// TIA Portal V20 export
TYPE "LBP_typeAlarmMsgs"
TITLE = PLC-Error / Messages / Erreur AP / messages
// User data type for block LBP_AlarmMessage [DB2] / Type de données utilisateur pour bloc LBP_AlarmMessage [DB2]
   STRUCT
      Chan : Array[1..10] of Struct   // From Channel 1..10 / Depuis canal 1..10
         FDD : Array[0..15] of Bool;   // Feed disable / Désactiver avance
         RID : Array[0..15] of Bool;   // Read-in disable / Désactiver importation
         NCSD : Array[0..15] of Bool;   // NC start disable / Désactiver Départ CN
         FdStop_1 : Array[0..15] of Bool;   // Feed stop GEOaxis 1 / Arrêt avance axe GEO 1
         FdStop_2 : Array[0..15] of Bool;   // Feed stop GEOaxis 2 / Arrêt avance axe GEO 2
         FdStop_3 : Array[0..15] of Bool;   // Feed stop GEOaxis 3 / Arrêt avance axe GEO 3
      END_STRUCT;
      Axis : Array[1..31] of Struct   // From Axis 1..31 / Depuis axe 1..31
         FdStop : Array[0..15] of Bool;   // Feed stop axis/spindle / Arrêt avance axe/broche
      END_STRUCT;
      AddValUserA0 : Array[0..63] of Int;   // Additional value for alarms in the user area 0 (700000..700063) / Valeur additionnelle pour les alarmes dans la zone utilisateur 0 (700000..700063)
      ChanA : Array[1..10] of Struct   // From Channel 1..10 / Depuis canal 1..10
         FDD_5C00xx : Array[0..15] of Bool;   // Feed disable Alarm no. 5C0000..5C0015 / Désactiver avance Alarme n° 5C0000..5C0015
         FDD_RID_5C01xx : Array[0..31] of Bool;   // Feed and read-in disable Alarm no. 5C0100..5C0131 / Désactiver avance et importation Alarme n° 5C0100..5C0131
         RID_5C02xx : Array[0..31] of Bool;   // Read-in disable Alarm no. 5C0200..5C0231 / Désactiver avance Alarme n° 5C0200..5C0231
         NCSD_5C03xx : Array[0..15] of Bool;   // NC start disable Alarm no. 5C0300..5C0315 / Désactiver Départ CN Alarme n° 5C0300..5C0315
         FdStop_1_5C11xx : Array[0..15] of Bool;   // Feed stop GEOaxis 1 Alarm no. 5C1100..5C1115 / Arrêt avance axe GEO 1 Alarme n° 5C1100..5C1115
         FdStop_2_5C12xx : Array[0..15] of Bool;   // Feed stop GEOaxis 2 Alarm no. 5C1200..5C1215 / Arrêt avance axe GEO 2 Alarme n° 5C1200..5C1215
         FdStop_3_5C13xx : Array[0..15] of Bool;   // Feed stop GEOaxis 3 Alarm no. 5C1300..5C1315 / Arrêt avance axe GEO 3 Alarme n° 5C1300..5C1315
      END_STRUCT;
      AxisA : Array[1..31] of Struct   // From Axis 1..31 / Depuis axe 1..31
         AAFdStop60AAxx : Array[0..15] of Bool;   // Feed stop axis/spindle / Arrêt avance axe/broche
      END_STRUCT;
      res552 : Word;   // Reserved / Réservé
      UserA : Array[0..63] of Struct
         A70UUxx : Array[0..63] of Bool;   // Alarm 70UU00..70UU63 (user area) / Alarme 70UU00..70UU63 (zone utilisateur)
      END_STRUCT;
   END_STRUCT;
   // // Chan[2].FDD : Feed disable / Désactiver avance
   // // Chan[3].FDD : Feed disable / Désactiver avance
   // // Chan[4].FDD : Feed disable / Désactiver avance
   // // Chan[5].FDD : Feed disable / Désactiver avance
   // // Chan[6].FDD : Feed disable / Désactiver avance
   // // Chan[7].FDD : Feed disable / Désactiver avance
   // // Chan[8].FDD : Feed disable / Désactiver avance
   // // Chan[9].FDD : Feed disable / Désactiver avance
   // // Chan[10].FDD : Feed disable / Désactiver avance
   // // Chan[2].RID : Read-in disable / Désactiver importation
   // // Chan[3].RID : Read-in disable / Désactiver importation
   // // Chan[4].RID : Read-in disable / Désactiver importation
   // // Chan[5].RID : Read-in disable / Désactiver importation
   // // Chan[6].RID : Read-in disable / Désactiver importation
   // // Chan[7].RID : Read-in disable / Désactiver importation
   // // Chan[8].RID : Read-in disable / Désactiver importation
   // // Chan[9].RID : Read-in disable / Désactiver importation
   // // Chan[10].RID : Read-in disable / Désactiver importation
   // // Chan[2].NCSD : NC start disable / Désactiver Départ CN
   // // Chan[3].NCSD : NC start disable / Désactiver Départ CN
   // // Chan[4].NCSD : NC start disable / Désactiver Départ CN
   // // Chan[5].NCSD : NC start disable / Désactiver Départ CN
   // // Chan[6].NCSD : NC start disable / Désactiver Départ CN
   // // Chan[7].NCSD : NC start disable / Désactiver Départ CN
   // // Chan[8].NCSD : NC start disable / Désactiver Départ CN
   // // Chan[9].NCSD : NC start disable / Désactiver Départ CN
   // // Chan[10].NCSD : NC start disable / Désactiver Départ CN
   // // Chan[2].FdStop_1 : Feed stop GEOaxis 1 / Arrêt avance axe GEO 1
   // // Chan[3].FdStop_1 : Feed stop GEOaxis 1 / Arrêt avance axe GEO 1
   // // Chan[4].FdStop_1 : Feed stop GEOaxis 1 / Arrêt avance axe GEO 1
   // // Chan[5].FdStop_1 : Feed stop GEOaxis 1 / Arrêt avance axe GEO 1
   // // Chan[6].FdStop_1 : Feed stop GEOaxis 1 / Arrêt avance axe GEO 1
   // // Chan[7].FdStop_1 : Feed stop GEOaxis 1 / Arrêt avance axe GEO 1
   // // Chan[8].FdStop_1 : Feed stop GEOaxis 1 / Arrêt avance axe GEO 1
   // // Chan[9].FdStop_1 : Feed stop GEOaxis 1 / Arrêt avance axe GEO 1
   // // Chan[10].FdStop_1 : Feed stop GEOaxis 1 / Arrêt avance axe GEO 1
   // // Chan[2].FdStop_2 : Feed stop GEOaxis 2 / Arrêt avance axe GEO 2
   // // Chan[3].FdStop_2 : Feed stop GEOaxis 2 / Arrêt avance axe GEO 2
   // // Chan[4].FdStop_2 : Feed stop GEOaxis 2 / Arrêt avance axe GEO 2
   // // Chan[5].FdStop_2 : Feed stop GEOaxis 2 / Arrêt avance axe GEO 2
   // // Chan[6].FdStop_2 : Feed stop GEOaxis 2 / Arrêt avance axe GEO 2
   // // Chan[7].FdStop_2 : Feed stop GEOaxis 2 / Arrêt avance axe GEO 2
   // // Chan[8].FdStop_2 : Feed stop GEOaxis 2 / Arrêt avance axe GEO 2
   // // Chan[9].FdStop_2 : Feed stop GEOaxis 2 / Arrêt avance axe GEO 2
   // // Chan[10].FdStop_2 : Feed stop GEOaxis 2 / Arrêt avance axe GEO 2
   // // Chan[2].FdStop_3 : Feed stop GEOaxis 3 / Arrêt avance axe GEO 3
   // // Chan[3].FdStop_3 : Feed stop GEOaxis 3 / Arrêt avance axe GEO 3
   // // Chan[4].FdStop_3 : Feed stop GEOaxis 3 / Arrêt avance axe GEO 3
   // // Chan[5].FdStop_3 : Feed stop GEOaxis 3 / Arrêt avance axe GEO 3
   // // Chan[6].FdStop_3 : Feed stop GEOaxis 3 / Arrêt avance axe GEO 3
   // // Chan[7].FdStop_3 : Feed stop GEOaxis 3 / Arrêt avance axe GEO 3
   // // Chan[8].FdStop_3 : Feed stop GEOaxis 3 / Arrêt avance axe GEO 3
   // // Chan[9].FdStop_3 : Feed stop GEOaxis 3 / Arrêt avance axe GEO 3
   // // Chan[10].FdStop_3 : Feed stop GEOaxis 3 / Arrêt avance axe GEO 3
   // // Chan[1] : From Channel 1..10 / Depuis canal 1..10
   // // Chan[2] : From Channel 1..10 / Depuis canal 1..10
   // // Chan[3] : From Channel 1..10 / Depuis canal 1..10
   // // Chan[4] : From Channel 1..10 / Depuis canal 1..10
   // // Chan[5] : From Channel 1..10 / Depuis canal 1..10
   // // Chan[6] : From Channel 1..10 / Depuis canal 1..10
   // // Chan[7] : From Channel 1..10 / Depuis canal 1..10
   // // Chan[8] : From Channel 1..10 / Depuis canal 1..10
   // // Chan[9] : From Channel 1..10 / Depuis canal 1..10
   // // Chan[10] : From Channel 1..10 / Depuis canal 1..10
   // // Axis[2].FdStop : Feed stop axis/spindle / Arrêt avance axe/broche
   // // Axis[3].FdStop : Feed stop axis/spindle / Arrêt avance axe/broche
   // // Axis[4].FdStop : Feed stop axis/spindle / Arrêt avance axe/broche
   // // Axis[5].FdStop : Feed stop axis/spindle / Arrêt avance axe/broche
   // // Axis[6].FdStop : Feed stop axis/spindle / Arrêt avance axe/broche
   // // Axis[7].FdStop : Feed stop axis/spindle / Arrêt avance axe/broche
   // // Axis[8].FdStop : Feed stop axis/spindle / Arrêt avance axe/broche
   // // Axis[9].FdStop : Feed stop axis/spindle / Arrêt avance axe/broche
   // // Axis[10].FdStop : Feed stop axis/spindle / Arrêt avance axe/broche
   // // Axis[11].FdStop : Feed stop axis/spindle / Arrêt avance axe/broche
   // // Axis[12].FdStop : Feed stop axis/spindle / Arrêt avance axe/broche
   // // Axis[13].FdStop : Feed stop axis/spindle / Arrêt avance axe/broche
   // // Axis[14].FdStop : Feed stop axis/spindle / Arrêt avance axe/broche
   // // Axis[15].FdStop : Feed stop axis/spindle / Arrêt avance axe/broche
   // // Axis[16].FdStop : Feed stop axis/spindle / Arrêt avance axe/broche
   // // Axis[17].FdStop : Feed stop axis/spindle / Arrêt avance axe/broche
   // // Axis[18].FdStop : Feed stop axis/spindle / Arrêt avance axe/broche
   // // Axis[19].FdStop : Feed stop axis/spindle / Arrêt avance axe/broche
   // // Axis[20].FdStop : Feed stop axis/spindle / Arrêt avance axe/broche
   // // Axis[21].FdStop : Feed stop axis/spindle / Arrêt avance axe/broche
   // // Axis[22].FdStop : Feed stop axis/spindle / Arrêt avance axe/broche
   // // Axis[23].FdStop : Feed stop axis/spindle / Arrêt avance axe/broche
   // // Axis[24].FdStop : Feed stop axis/spindle / Arrêt avance axe/broche
   // // Axis[25].FdStop : Feed stop axis/spindle / Arrêt avance axe/broche
   // // Axis[26].FdStop : Feed stop axis/spindle / Arrêt avance axe/broche
   // // Axis[27].FdStop : Feed stop axis/spindle / Arrêt avance axe/broche
   // // Axis[28].FdStop : Feed stop axis/spindle / Arrêt avance axe/broche
   // // Axis[29].FdStop : Feed stop axis/spindle / Arrêt avance axe/broche
   // // Axis[30].FdStop : Feed stop axis/spindle / Arrêt avance axe/broche
   // // Axis[31].FdStop : Feed stop axis/spindle / Arrêt avance axe/broche
   // // Axis[1] : From Axis 1..31 / Depuis axe 1..31
   // // Axis[2] : From Axis 1..31 / Depuis axe 1..31
   // // Axis[3] : From Axis 1..31 / Depuis axe 1..31
   // // Axis[4] : From Axis 1..31 / Depuis axe 1..31
   // // Axis[5] : From Axis 1..31 / Depuis axe 1..31
   // // Axis[6] : From Axis 1..31 / Depuis axe 1..31
   // // Axis[7] : From Axis 1..31 / Depuis axe 1..31
   // // Axis[8] : From Axis 1..31 / Depuis axe 1..31
   // // Axis[9] : From Axis 1..31 / Depuis axe 1..31
   // // Axis[10] : From Axis 1..31 / Depuis axe 1..31
   // // Axis[11] : From Axis 1..31 / Depuis axe 1..31
   // // Axis[12] : From Axis 1..31 / Depuis axe 1..31
   // // Axis[13] : From Axis 1..31 / Depuis axe 1..31
   // // Axis[14] : From Axis 1..31 / Depuis axe 1..31
   // // Axis[15] : From Axis 1..31 / Depuis axe 1..31
   // // Axis[16] : From Axis 1..31 / Depuis axe 1..31
   // // Axis[17] : From Axis 1..31 / Depuis axe 1..31
   // // Axis[18] : From Axis 1..31 / Depuis axe 1..31
   // // Axis[19] : From Axis 1..31 / Depuis axe 1..31
   // // Axis[20] : From Axis 1..31 / Depuis axe 1..31
   // // Axis[21] : From Axis 1..31 / Depuis axe 1..31
   // // Axis[22] : From Axis 1..31 / Depuis axe 1..31
   // // Axis[23] : From Axis 1..31 / Depuis axe 1..31
   // // Axis[24] : From Axis 1..31 / Depuis axe 1..31
   // // Axis[25] : From Axis 1..31 / Depuis axe 1..31
   // // Axis[26] : From Axis 1..31 / Depuis axe 1..31
   // // Axis[27] : From Axis 1..31 / Depuis axe 1..31
   // // Axis[28] : From Axis 1..31 / Depuis axe 1..31
   // // Axis[29] : From Axis 1..31 / Depuis axe 1..31
   // // Axis[30] : From Axis 1..31 / Depuis axe 1..31
   // // Axis[31] : From Axis 1..31 / Depuis axe 1..31
   // // ChanA[2].FDD_5C00xx : Feed disable Alarm no. 5C0000..5C0015 / Désactiver avance Alarme n° 5C0000..5C0015
   // // ChanA[3].FDD_5C00xx : Feed disable Alarm no. 5C0000..5C0015 / Désactiver avance Alarme n° 5C0000..5C0015
   // // ChanA[4].FDD_5C00xx : Feed disable Alarm no. 5C0000..5C0015 / Désactiver avance Alarme n° 5C0000..5C0015
   // // ChanA[5].FDD_5C00xx : Feed disable Alarm no. 5C0000..5C0015 / Désactiver avance Alarme n° 5C0000..5C0015
   // // ChanA[6].FDD_5C00xx : Feed disable Alarm no. 5C0000..5C0015 / Désactiver avance Alarme n° 5C0000..5C0015
   // // ChanA[7].FDD_5C00xx : Feed disable Alarm no. 5C0000..5C0015 / Désactiver avance Alarme n° 5C0000..5C0015
   // // ChanA[8].FDD_5C00xx : Feed disable Alarm no. 5C0000..5C0015 / Désactiver avance Alarme n° 5C0000..5C0015
   // // ChanA[9].FDD_5C00xx : Feed disable Alarm no. 5C0000..5C0015 / Désactiver avance Alarme n° 5C0000..5C0015
   // // ChanA[10].FDD_5C00xx : Feed disable Alarm no. 5C0000..5C0015 / Désactiver avance Alarme n° 5C0000..5C0015
   // // ChanA[2].FDD_RID_5C01xx : Feed and read-in disable Alarm no. 5C0100..5C0131 / Désactiver avance et importation Alarme n° 5C0100..5C0131
   // // ChanA[3].FDD_RID_5C01xx : Feed and read-in disable Alarm no. 5C0100..5C0131 / Désactiver avance et importation Alarme n° 5C0100..5C0131
   // // ChanA[4].FDD_RID_5C01xx : Feed and read-in disable Alarm no. 5C0100..5C0131 / Désactiver avance et importation Alarme n° 5C0100..5C0131
   // // ChanA[5].FDD_RID_5C01xx : Feed and read-in disable Alarm no. 5C0100..5C0131 / Désactiver avance et importation Alarme n° 5C0100..5C0131
   // // ChanA[6].FDD_RID_5C01xx : Feed and read-in disable Alarm no. 5C0100..5C0131 / Désactiver avance et importation Alarme n° 5C0100..5C0131
   // // ChanA[7].FDD_RID_5C01xx : Feed and read-in disable Alarm no. 5C0100..5C0131 / Désactiver avance et importation Alarme n° 5C0100..5C0131
   // // ChanA[8].FDD_RID_5C01xx : Feed and read-in disable Alarm no. 5C0100..5C0131 / Désactiver avance et importation Alarme n° 5C0100..5C0131
   // // ChanA[9].FDD_RID_5C01xx : Feed and read-in disable Alarm no. 5C0100..5C0131 / Désactiver avance et importation Alarme n° 5C0100..5C0131
   // // ChanA[10].FDD_RID_5C01xx : Feed and read-in disable Alarm no. 5C0100..5C0131 / Désactiver avance et importation Alarme n° 5C0100..5C0131
   // // ChanA[2].RID_5C02xx : Read-in disable Alarm no. 5C0200..5C0231 / Désactiver avance Alarme n° 5C0200..5C0231
   // // ChanA[3].RID_5C02xx : Read-in disable Alarm no. 5C0200..5C0231 / Désactiver avance Alarme n° 5C0200..5C0231
   // // ChanA[4].RID_5C02xx : Read-in disable Alarm no. 5C0200..5C0231 / Désactiver avance Alarme n° 5C0200..5C0231
   // // ChanA[5].RID_5C02xx : Read-in disable Alarm no. 5C0200..5C0231 / Désactiver avance Alarme n° 5C0200..5C0231
   // // ChanA[6].RID_5C02xx : Read-in disable Alarm no. 5C0200..5C0231 / Désactiver avance Alarme n° 5C0200..5C0231
   // // ChanA[7].RID_5C02xx : Read-in disable Alarm no. 5C0200..5C0231 / Désactiver avance Alarme n° 5C0200..5C0231
   // // ChanA[8].RID_5C02xx : Read-in disable Alarm no. 5C0200..5C0231 / Désactiver avance Alarme n° 5C0200..5C0231
   // // ChanA[9].RID_5C02xx : Read-in disable Alarm no. 5C0200..5C0231 / Désactiver avance Alarme n° 5C0200..5C0231
   // // ChanA[10].RID_5C02xx : Read-in disable Alarm no. 5C0200..5C0231 / Désactiver avance Alarme n° 5C0200..5C0231
   // // ChanA[2].NCSD_5C03xx : NC start disable Alarm no. 5C0300..5C0315 / Désactiver Départ CN Alarme n° 5C0300..5C0315
   // // ChanA[3].NCSD_5C03xx : NC start disable Alarm no. 5C0300..5C0315 / Désactiver Départ CN Alarme n° 5C0300..5C0315
   // // ChanA[4].NCSD_5C03xx : NC start disable Alarm no. 5C0300..5C0315 / Désactiver Départ CN Alarme n° 5C0300..5C0315
   // // ChanA[5].NCSD_5C03xx : NC start disable Alarm no. 5C0300..5C0315 / Désactiver Départ CN Alarme n° 5C0300..5C0315
   // // ChanA[6].NCSD_5C03xx : NC start disable Alarm no. 5C0300..5C0315 / Désactiver Départ CN Alarme n° 5C0300..5C0315
   // // ChanA[7].NCSD_5C03xx : NC start disable Alarm no. 5C0300..5C0315 / Désactiver Départ CN Alarme n° 5C0300..5C0315
   // // ChanA[8].NCSD_5C03xx : NC start disable Alarm no. 5C0300..5C0315 / Désactiver Départ CN Alarme n° 5C0300..5C0315
   // // ChanA[9].NCSD_5C03xx : NC start disable Alarm no. 5C0300..5C0315 / Désactiver Départ CN Alarme n° 5C0300..5C0315
   // // ChanA[10].NCSD_5C03xx : NC start disable Alarm no. 5C0300..5C0315 / Désactiver Départ CN Alarme n° 5C0300..5C0315
   // // ChanA[2].FdStop_1_5C11xx : Feed stop GEOaxis 1 Alarm no. 5C1100..5C1115 / Arrêt avance axe GEO 1 Alarme n° 5C1100..5C1115
   // // ChanA[3].FdStop_1_5C11xx : Feed stop GEOaxis 1 Alarm no. 5C1100..5C1115 / Arrêt avance axe GEO 1 Alarme n° 5C1100..5C1115
   // // ChanA[4].FdStop_1_5C11xx : Feed stop GEOaxis 1 Alarm no. 5C1100..5C1115 / Arrêt avance axe GEO 1 Alarme n° 5C1100..5C1115
   // // ChanA[5].FdStop_1_5C11xx : Feed stop GEOaxis 1 Alarm no. 5C1100..5C1115 / Arrêt avance axe GEO 1 Alarme n° 5C1100..5C1115
   // // ChanA[6].FdStop_1_5C11xx : Feed stop GEOaxis 1 Alarm no. 5C1100..5C1115 / Arrêt avance axe GEO 1 Alarme n° 5C1100..5C1115
   // // ChanA[7].FdStop_1_5C11xx : Feed stop GEOaxis 1 Alarm no. 5C1100..5C1115 / Arrêt avance axe GEO 1 Alarme n° 5C1100..5C1115
   // // ChanA[8].FdStop_1_5C11xx : Feed stop GEOaxis 1 Alarm no. 5C1100..5C1115 / Arrêt avance axe GEO 1 Alarme n° 5C1100..5C1115
   // // ChanA[9].FdStop_1_5C11xx : Feed stop GEOaxis 1 Alarm no. 5C1100..5C1115 / Arrêt avance axe GEO 1 Alarme n° 5C1100..5C1115
   // // ChanA[10].FdStop_1_5C11xx : Feed stop GEOaxis 1 Alarm no. 5C1100..5C1115 / Arrêt avance axe GEO 1 Alarme n° 5C1100..5C1115
   // // ChanA[2].FdStop_2_5C12xx : Feed stop GEOaxis 2 Alarm no. 5C1200..5C1215 / Arrêt avance axe GEO 2 Alarme n° 5C1200..5C1215
   // // ChanA[3].FdStop_2_5C12xx : Feed stop GEOaxis 2 Alarm no. 5C1200..5C1215 / Arrêt avance axe GEO 2 Alarme n° 5C1200..5C1215
   // // ChanA[4].FdStop_2_5C12xx : Feed stop GEOaxis 2 Alarm no. 5C1200..5C1215 / Arrêt avance axe GEO 2 Alarme n° 5C1200..5C1215
   // // ChanA[5].FdStop_2_5C12xx : Feed stop GEOaxis 2 Alarm no. 5C1200..5C1215 / Arrêt avance axe GEO 2 Alarme n° 5C1200..5C1215
   // // ChanA[6].FdStop_2_5C12xx : Feed stop GEOaxis 2 Alarm no. 5C1200..5C1215 / Arrêt avance axe GEO 2 Alarme n° 5C1200..5C1215
   // // ChanA[7].FdStop_2_5C12xx : Feed stop GEOaxis 2 Alarm no. 5C1200..5C1215 / Arrêt avance axe GEO 2 Alarme n° 5C1200..5C1215
   // // ChanA[8].FdStop_2_5C12xx : Feed stop GEOaxis 2 Alarm no. 5C1200..5C1215 / Arrêt avance axe GEO 2 Alarme n° 5C1200..5C1215
   // // ChanA[9].FdStop_2_5C12xx : Feed stop GEOaxis 2 Alarm no. 5C1200..5C1215 / Arrêt avance axe GEO 2 Alarme n° 5C1200..5C1215
   // // ChanA[10].FdStop_2_5C12xx : Feed stop GEOaxis 2 Alarm no. 5C1200..5C1215 / Arrêt avance axe GEO 2 Alarme n° 5C1200..5C1215
   // // ChanA[2].FdStop_3_5C13xx : Feed stop GEOaxis 3 Alarm no. 5C1300..5C1315 / Arrêt avance axe GEO 3 Alarme n° 5C1300..5C1315
   // // ChanA[3].FdStop_3_5C13xx : Feed stop GEOaxis 3 Alarm no. 5C1300..5C1315 / Arrêt avance axe GEO 3 Alarme n° 5C1300..5C1315
   // // ChanA[4].FdStop_3_5C13xx : Feed stop GEOaxis 3 Alarm no. 5C1300..5C1315 / Arrêt avance axe GEO 3 Alarme n° 5C1300..5C1315
   // // ChanA[5].FdStop_3_5C13xx : Feed stop GEOaxis 3 Alarm no. 5C1300..5C1315 / Arrêt avance axe GEO 3 Alarme n° 5C1300..5C1315
   // // ChanA[6].FdStop_3_5C13xx : Feed stop GEOaxis 3 Alarm no. 5C1300..5C1315 / Arrêt avance axe GEO 3 Alarme n° 5C1300..5C1315
   // // ChanA[7].FdStop_3_5C13xx : Feed stop GEOaxis 3 Alarm no. 5C1300..5C1315 / Arrêt avance axe GEO 3 Alarme n° 5C1300..5C1315
   // // ChanA[8].FdStop_3_5C13xx : Feed stop GEOaxis 3 Alarm no. 5C1300..5C1315 / Arrêt avance axe GEO 3 Alarme n° 5C1300..5C1315
   // // ChanA[9].FdStop_3_5C13xx : Feed stop GEOaxis 3 Alarm no. 5C1300..5C1315 / Arrêt avance axe GEO 3 Alarme n° 5C1300..5C1315
   // // ChanA[10].FdStop_3_5C13xx : Feed stop GEOaxis 3 Alarm no. 5C1300..5C1315 / Arrêt avance axe GEO 3 Alarme n° 5C1300..5C1315
   // // ChanA[1] : From Channel 1..10 / Depuis canal 1..10
   // // ChanA[2] : From Channel 1..10 / Depuis canal 1..10
   // // ChanA[3] : From Channel 1..10 / Depuis canal 1..10
   // // ChanA[4] : From Channel 1..10 / Depuis canal 1..10
   // // ChanA[5] : From Channel 1..10 / Depuis canal 1..10
   // // ChanA[6] : From Channel 1..10 / Depuis canal 1..10
   // // ChanA[7] : From Channel 1..10 / Depuis canal 1..10
   // // ChanA[8] : From Channel 1..10 / Depuis canal 1..10
   // // ChanA[9] : From Channel 1..10 / Depuis canal 1..10
   // // ChanA[10] : From Channel 1..10 / Depuis canal 1..10
   // // AxisA[2].AAFdStop60AAxx : Feed stop axis/spindle / Arrêt avance axe/broche
   // // AxisA[3].AAFdStop60AAxx : Feed stop axis/spindle / Arrêt avance axe/broche
   // // AxisA[4].AAFdStop60AAxx : Feed stop axis/spindle / Arrêt avance axe/broche
   // // AxisA[5].AAFdStop60AAxx : Feed stop axis/spindle / Arrêt avance axe/broche
   // // AxisA[6].AAFdStop60AAxx : Feed stop axis/spindle / Arrêt avance axe/broche
   // // AxisA[7].AAFdStop60AAxx : Feed stop axis/spindle / Arrêt avance axe/broche
   // // AxisA[8].AAFdStop60AAxx : Feed stop axis/spindle / Arrêt avance axe/broche
   // // AxisA[9].AAFdStop60AAxx : Feed stop axis/spindle / Arrêt avance axe/broche
   // // AxisA[10].AAFdStop60AAxx : Feed stop axis/spindle / Arrêt avance axe/broche
   // // AxisA[11].AAFdStop60AAxx : Feed stop axis/spindle / Arrêt avance axe/broche
   // // AxisA[12].AAFdStop60AAxx : Feed stop axis/spindle / Arrêt avance axe/broche
   // // AxisA[13].AAFdStop60AAxx : Feed stop axis/spindle / Arrêt avance axe/broche
   // // AxisA[14].AAFdStop60AAxx : Feed stop axis/spindle / Arrêt avance axe/broche
   // // AxisA[15].AAFdStop60AAxx : Feed stop axis/spindle / Arrêt avance axe/broche
   // // AxisA[16].AAFdStop60AAxx : Feed stop axis/spindle / Arrêt avance axe/broche
   // // AxisA[17].AAFdStop60AAxx : Feed stop axis/spindle / Arrêt avance axe/broche
   // // AxisA[18].AAFdStop60AAxx : Feed stop axis/spindle / Arrêt avance axe/broche
   // // AxisA[19].AAFdStop60AAxx : Feed stop axis/spindle / Arrêt avance axe/broche
   // // AxisA[20].AAFdStop60AAxx : Feed stop axis/spindle / Arrêt avance axe/broche
   // // AxisA[21].AAFdStop60AAxx : Feed stop axis/spindle / Arrêt avance axe/broche
   // // AxisA[22].AAFdStop60AAxx : Feed stop axis/spindle / Arrêt avance axe/broche
   // // AxisA[23].AAFdStop60AAxx : Feed stop axis/spindle / Arrêt avance axe/broche
   // // AxisA[24].AAFdStop60AAxx : Feed stop axis/spindle / Arrêt avance axe/broche
   // // AxisA[25].AAFdStop60AAxx : Feed stop axis/spindle / Arrêt avance axe/broche
   // // AxisA[26].AAFdStop60AAxx : Feed stop axis/spindle / Arrêt avance axe/broche
   // // AxisA[27].AAFdStop60AAxx : Feed stop axis/spindle / Arrêt avance axe/broche
   // // AxisA[28].AAFdStop60AAxx : Feed stop axis/spindle / Arrêt avance axe/broche
   // // AxisA[29].AAFdStop60AAxx : Feed stop axis/spindle / Arrêt avance axe/broche
   // // AxisA[30].AAFdStop60AAxx : Feed stop axis/spindle / Arrêt avance axe/broche
   // // AxisA[31].AAFdStop60AAxx : Feed stop axis/spindle / Arrêt avance axe/broche
   // // AxisA[1] : From Axis 1..31 / Depuis axe 1..31
   // // AxisA[2] : From Axis 1..31 / Depuis axe 1..31
   // // AxisA[3] : From Axis 1..31 / Depuis axe 1..31
   // // AxisA[4] : From Axis 1..31 / Depuis axe 1..31
   // // AxisA[5] : From Axis 1..31 / Depuis axe 1..31
   // // AxisA[6] : From Axis 1..31 / Depuis axe 1..31
   // // AxisA[7] : From Axis 1..31 / Depuis axe 1..31
   // // AxisA[8] : From Axis 1..31 / Depuis axe 1..31
   // // AxisA[9] : From Axis 1..31 / Depuis axe 1..31
   // // AxisA[10] : From Axis 1..31 / Depuis axe 1..31
   // // AxisA[11] : From Axis 1..31 / Depuis axe 1..31
   // // AxisA[12] : From Axis 1..31 / Depuis axe 1..31
   // // AxisA[13] : From Axis 1..31 / Depuis axe 1..31
   // // AxisA[14] : From Axis 1..31 / Depuis axe 1..31
   // // AxisA[15] : From Axis 1..31 / Depuis axe 1..31
   // // AxisA[16] : From Axis 1..31 / Depuis axe 1..31
   // // AxisA[17] : From Axis 1..31 / Depuis axe 1..31
   // // AxisA[18] : From Axis 1..31 / Depuis axe 1..31
   // // AxisA[19] : From Axis 1..31 / Depuis axe 1..31
   // // AxisA[20] : From Axis 1..31 / Depuis axe 1..31
   // // AxisA[21] : From Axis 1..31 / Depuis axe 1..31
   // // AxisA[22] : From Axis 1..31 / Depuis axe 1..31
   // // AxisA[23] : From Axis 1..31 / Depuis axe 1..31
   // // AxisA[24] : From Axis 1..31 / Depuis axe 1..31
   // // AxisA[25] : From Axis 1..31 / Depuis axe 1..31
   // // AxisA[26] : From Axis 1..31 / Depuis axe 1..31
   // // AxisA[27] : From Axis 1..31 / Depuis axe 1..31
   // // AxisA[28] : From Axis 1..31 / Depuis axe 1..31
   // // AxisA[29] : From Axis 1..31 / Depuis axe 1..31
   // // AxisA[30] : From Axis 1..31 / Depuis axe 1..31
   // // AxisA[31] : From Axis 1..31 / Depuis axe 1..31
   // // UserA[1].A70UUxx : Alarm 70UU00..70UU63 (user area) / Alarme 70UU00..70UU63 (zone utilisateur)
   // // UserA[2].A70UUxx : Alarm 70UU00..70UU63 (user area) / Alarme 70UU00..70UU63 (zone utilisateur)
   // // UserA[3].A70UUxx : Alarm 70UU00..70UU63 (user area) / Alarme 70UU00..70UU63 (zone utilisateur)
   // // UserA[4].A70UUxx : Alarm 70UU00..70UU63 (user area) / Alarme 70UU00..70UU63 (zone utilisateur)
   // // UserA[5].A70UUxx : Alarm 70UU00..70UU63 (user area) / Alarme 70UU00..70UU63 (zone utilisateur)
   // // UserA[6].A70UUxx : Alarm 70UU00..70UU63 (user area) / Alarme 70UU00..70UU63 (zone utilisateur)
   // // UserA[7].A70UUxx : Alarm 70UU00..70UU63 (user area) / Alarme 70UU00..70UU63 (zone utilisateur)
   // // UserA[8].A70UUxx : Alarm 70UU00..70UU63 (user area) / Alarme 70UU00..70UU63 (zone utilisateur)
   // // UserA[9].A70UUxx : Alarm 70UU00..70UU63 (user area) / Alarme 70UU00..70UU63 (zone utilisateur)
   // // UserA[10].A70UUxx : Alarm 70UU00..70UU63 (user area) / Alarme 70UU00..70UU63 (zone utilisateur)
   // // UserA[11].A70UUxx : Alarm 70UU00..70UU63 (user area) / Alarme 70UU00..70UU63 (zone utilisateur)
   // // UserA[12].A70UUxx : Alarm 70UU00..70UU63 (user area) / Alarme 70UU00..70UU63 (zone utilisateur)
   // // UserA[13].A70UUxx : Alarm 70UU00..70UU63 (user area) / Alarme 70UU00..70UU63 (zone utilisateur)
   // // UserA[14].A70UUxx : Alarm 70UU00..70UU63 (user area) / Alarme 70UU00..70UU63 (zone utilisateur)
   // // UserA[15].A70UUxx : Alarm 70UU00..70UU63 (user area) / Alarme 70UU00..70UU63 (zone utilisateur)
   // // UserA[16].A70UUxx : Alarm 70UU00..70UU63 (user area) / Alarme 70UU00..70UU63 (zone utilisateur)
   // // UserA[17].A70UUxx : Alarm 70UU00..70UU63 (user area) / Alarme 70UU00..70UU63 (zone utilisateur)
   // // UserA[18].A70UUxx : Alarm 70UU00..70UU63 (user area) / Alarme 70UU00..70UU63 (zone utilisateur)
   // // UserA[19].A70UUxx : Alarm 70UU00..70UU63 (user area) / Alarme 70UU00..70UU63 (zone utilisateur)
   // // UserA[20].A70UUxx : Alarm 70UU00..70UU63 (user area) / Alarme 70UU00..70UU63 (zone utilisateur)
   // // UserA[21].A70UUxx : Alarm 70UU00..70UU63 (user area) / Alarme 70UU00..70UU63 (zone utilisateur)
   // // UserA[22].A70UUxx : Alarm 70UU00..70UU63 (user area) / Alarme 70UU00..70UU63 (zone utilisateur)
   // // UserA[23].A70UUxx : Alarm 70UU00..70UU63 (user area) / Alarme 70UU00..70UU63 (zone utilisateur)
   // // UserA[24].A70UUxx : Alarm 70UU00..70UU63 (user area) / Alarme 70UU00..70UU63 (zone utilisateur)
   // // UserA[25].A70UUxx : Alarm 70UU00..70UU63 (user area) / Alarme 70UU00..70UU63 (zone utilisateur)
   // // UserA[26].A70UUxx : Alarm 70UU00..70UU63 (user area) / Alarme 70UU00..70UU63 (zone utilisateur)
   // // UserA[27].A70UUxx : Alarm 70UU00..70UU63 (user area) / Alarme 70UU00..70UU63 (zone utilisateur)
   // // UserA[28].A70UUxx : Alarm 70UU00..70UU63 (user area) / Alarme 70UU00..70UU63 (zone utilisateur)
   // // UserA[29].A70UUxx : Alarm 70UU00..70UU63 (user area) / Alarme 70UU00..70UU63 (zone utilisateur)
   // // UserA[30].A70UUxx : Alarm 70UU00..70UU63 (user area) / Alarme 70UU00..70UU63 (zone utilisateur)
   // // UserA[31].A70UUxx : Alarm 70UU00..70UU63 (user area) / Alarme 70UU00..70UU63 (zone utilisateur)
   // // UserA[32].A70UUxx : Alarm 70UU00..70UU63 (user area) / Alarme 70UU00..70UU63 (zone utilisateur)
   // // UserA[33].A70UUxx : Alarm 70UU00..70UU63 (user area) / Alarme 70UU00..70UU63 (zone utilisateur)
   // // UserA[34].A70UUxx : Alarm 70UU00..70UU63 (user area) / Alarme 70UU00..70UU63 (zone utilisateur)
   // // UserA[35].A70UUxx : Alarm 70UU00..70UU63 (user area) / Alarme 70UU00..70UU63 (zone utilisateur)
   // // UserA[36].A70UUxx : Alarm 70UU00..70UU63 (user area) / Alarme 70UU00..70UU63 (zone utilisateur)
   // // UserA[37].A70UUxx : Alarm 70UU00..70UU63 (user area) / Alarme 70UU00..70UU63 (zone utilisateur)
   // // UserA[38].A70UUxx : Alarm 70UU00..70UU63 (user area) / Alarme 70UU00..70UU63 (zone utilisateur)
   // // UserA[39].A70UUxx : Alarm 70UU00..70UU63 (user area) / Alarme 70UU00..70UU63 (zone utilisateur)
   // // UserA[40].A70UUxx : Alarm 70UU00..70UU63 (user area) / Alarme 70UU00..70UU63 (zone utilisateur)
   // // UserA[41].A70UUxx : Alarm 70UU00..70UU63 (user area) / Alarme 70UU00..70UU63 (zone utilisateur)
   // // UserA[42].A70UUxx : Alarm 70UU00..70UU63 (user area) / Alarme 70UU00..70UU63 (zone utilisateur)
   // // UserA[43].A70UUxx : Alarm 70UU00..70UU63 (user area) / Alarme 70UU00..70UU63 (zone utilisateur)
   // // UserA[44].A70UUxx : Alarm 70UU00..70UU63 (user area) / Alarme 70UU00..70UU63 (zone utilisateur)
   // // UserA[45].A70UUxx : Alarm 70UU00..70UU63 (user area) / Alarme 70UU00..70UU63 (zone utilisateur)
   // // UserA[46].A70UUxx : Alarm 70UU00..70UU63 (user area) / Alarme 70UU00..70UU63 (zone utilisateur)
   // // UserA[47].A70UUxx : Alarm 70UU00..70UU63 (user area) / Alarme 70UU00..70UU63 (zone utilisateur)
   // // UserA[48].A70UUxx : Alarm 70UU00..70UU63 (user area) / Alarme 70UU00..70UU63 (zone utilisateur)
   // // UserA[49].A70UUxx : Alarm 70UU00..70UU63 (user area) / Alarme 70UU00..70UU63 (zone utilisateur)
   // // UserA[50].A70UUxx : Alarm 70UU00..70UU63 (user area) / Alarme 70UU00..70UU63 (zone utilisateur)
   // // UserA[51].A70UUxx : Alarm 70UU00..70UU63 (user area) / Alarme 70UU00..70UU63 (zone utilisateur)
   // // UserA[52].A70UUxx : Alarm 70UU00..70UU63 (user area) / Alarme 70UU00..70UU63 (zone utilisateur)
   // // UserA[53].A70UUxx : Alarm 70UU00..70UU63 (user area) / Alarme 70UU00..70UU63 (zone utilisateur)
   // // UserA[54].A70UUxx : Alarm 70UU00..70UU63 (user area) / Alarme 70UU00..70UU63 (zone utilisateur)
   // // UserA[55].A70UUxx : Alarm 70UU00..70UU63 (user area) / Alarme 70UU00..70UU63 (zone utilisateur)
   // // UserA[56].A70UUxx : Alarm 70UU00..70UU63 (user area) / Alarme 70UU00..70UU63 (zone utilisateur)
   // // UserA[57].A70UUxx : Alarm 70UU00..70UU63 (user area) / Alarme 70UU00..70UU63 (zone utilisateur)
   // // UserA[58].A70UUxx : Alarm 70UU00..70UU63 (user area) / Alarme 70UU00..70UU63 (zone utilisateur)
   // // UserA[59].A70UUxx : Alarm 70UU00..70UU63 (user area) / Alarme 70UU00..70UU63 (zone utilisateur)
   // // UserA[60].A70UUxx : Alarm 70UU00..70UU63 (user area) / Alarme 70UU00..70UU63 (zone utilisateur)
   // // UserA[61].A70UUxx : Alarm 70UU00..70UU63 (user area) / Alarme 70UU00..70UU63 (zone utilisateur)
   // // UserA[62].A70UUxx : Alarm 70UU00..70UU63 (user area) / Alarme 70UU00..70UU63 (zone utilisateur)
   // // UserA[63].A70UUxx : Alarm 70UU00..70UU63 (user area) / Alarme 70UU00..70UU63 (zone utilisateur)
END_TYPE
